Universal Robots PolyScope program: DynamicAxisPositionCheck.urp

ProgramRoot directory=/home/ur/ursim-3.1/programs/Howtos; kinematics=(a=[0, -0.425, -0.39225, 0, 0, 0], d=[0.08916, 0, 0, 0.10915, 0.09465, 0.0823], alpha=[1.5708, 0, 0, 1.5708, -1.5708, 0], deltaTheta=[0, 0, 0, 0, 0, 0], status=notInitialized); lastSavedInVersion=(project__name=Polyscope, major__version=3, minor__version=1, svn__revision=17195, build__date=Mar 11 2015, 13:02:28); name=DynamicAxisPositionCheck; programVersion=(project__name=Polyscope, major__version=3, minor__version=1, svn__revision=17195, build__date=Mar 11 2015, 13:02:28); robotEnvironmentFileName=default; serialNumberRobot=2014350001
  MainProgram cartesianAcceleration=1.2; cartesianSpeed=0.25; jointAcceleration=1.3962634015954636; jointSpeed=1.0471975511965976; sharedProcessMoveBlendRadius=0.025; motionType=JOINT_SPACE
    Move cartesianAcceleration=1.2; cartesianSpeed=0.25; jointAcceleration=1.3962634015954636; jointSpeed=1.0471975511965976; sharedProcessMoveBlendRadius=0.025; motionType=JOINT_SPACE
      Waypoint blendRadius=0.05; cartesianAcceleration=1.2; cartesianSpeed=0.25; jointAcceleration=1.3962634015954636; jointSpeed=1.0471975511965976; nextMotionTime=2.0; stoppoint=true; useSharedBlendParameter=true; useSharedParameters=true; position=TCP in base x=-120.113 y=-431.763 z=146.073 mm, rx=-0.0012 ry=3.1163 rz=0.0389 rad; joints [-91.713, -98.956, -126.223, -46.295, 91.393, -1.776] deg; positionType=FIXED_POSITION; waypointPoseInFeatureCoordinates=(pos=(x=-0.12011317028458361, y=-0.4317631667637431, z=0.14607252291477704), rot=(x=-0.0012209830284081382, y=3.1162764812408743, z=0.03889191616813277)); name=Waypoint_1
      Waypoint blendRadius=0.05; cartesianAcceleration=1.2; cartesianSpeed=0.25; jointAcceleration=1.3962634015954636; jointSpeed=1.0471975511965976; nextMotionTime=2.0; stoppoint=true; useSharedBlendParameter=true; useSharedParameters=true; position=TCP in base x=445.565 y=48.146 z=146.073 mm, rx=2.5949 ry=-1.7583 rz=-0.0545 rad; joints [20, -98.956, -126.223, -46.295, 91.393, -1.776] deg; positionType=FIXED_POSITION; waypointPoseInFeatureCoordinates=(pos=(x=0.44556545780559137, y=0.04814591010836716, z=0.14607252291477704), rot=(x=2.5949451445964606, y=-1.7582886681424552, z=-0.05448402614874925)); name=Waypoint_2
  Thread name=Thread_1
    Assignment expr=get_actual_joint_positions(); operatorValueType=INTEGER; valueSource=EXPRESSION
    Assignment expr=ExpressionVariableNode[0]; operatorValueType=INTEGER; valueSource=EXPRESSION
    If expr=ExpressionVariableNode>0; type=IF_NODE
      Set 
    If type=ELSE_NODE
      Set 
    Script type=0; expressionBranchNode=sync()
